// TIA Portal V17 export
// export: Created 2023-02-14T02:49:50.4456623Z, ExportSetting WithDefaults, DisplayName Totally Integrated Automation Portal, DisplayVersion V17, DisplayName TIA Portal Openness, DisplayVersion V17, DisplayName TIA Portal Teamcenter Gateway, DisplayVersion V17, DisplayName TIA Portal Version Control Interface, DisplayVersion V17, DisplayName SINAMICS Startdrive Advanced, DisplayVersion V17, DisplayName SINAMICS Startdrive G130, G150, S120, S150, SINAMICS MV, S210, DisplayVersion V17, DisplayName SINAMICS Startdrive G110M, G120, G120C, G120D, G120P, G115D, DisplayVersion V17, DisplayName STEP 7 Professional, DisplayVersion V17, DisplayName STEP 7 Safety, DisplayVersion V17, DisplayName WinCC Professional, DisplayVersion V17
DATA_BLOCK "T-05.01_DB"   // DB355
VERSION : 0.1
// stored: AutoNumber false, DBAccessibleFromOPCUA true, DBAccessibleFromWebserver true, InstanceOfName BFT_Type2, InstanceOfType FB
"BFT_Type2"
   // VAR_INPUT
   //    "IN_FBAV.01" : Bool;
   //    "IN_FBAV.02" : Bool;
   //    "IN_FBAV.03" : Bool;
   //    "IN_FBAV.04" : Bool;
   //    "IN_FBAV.05" : Bool;
   //    "IN_FBAV.06" : Bool;
   //    "IN_FBAV.07" : Bool;
   //    "IN_FBAV.08" : Bool;
   //    "IN_FBAV.09" : Bool;
   //    "IN_FBAV.10" : Bool;
   //    "IN_FBAV.11" : Bool;
   //    "IN_FBAV.12" : Bool;
   //    IN_LT01 : Real;
   //    "IN_FBP.01" : Bool;
   //    "IN_P.01-Speed" : Real;
   //    "IN_FBP.02" : Bool;
   //    "IN_P.02-Speed" : Real;
   //    "IN_FBP.03" : Bool;
   //    "IN_P.03-Speed" : Real;
   //    IN_FBXA : Bool;
   //    "IN_XA-Speed" : Real;
   //    DosePumpSpeed : Real;
   //    "DoseON-OFF" : Bool;
   //    "DosePumpON-OFF" : Bool;
   //    CIPPulse : Bool;
   //    CIP_Supply_ON : Bool;
   //    CIP_Busy : Bool;
   //    LineTrf_OK : Bool;
   //    LineFlush_OK : Bool;
   //    Loading_Busy : Bool;
   //    LCS_Start : Bool;
   //    LCS_Stop : Bool;
   //    LCS_Dose : Bool;
   //    InloadDose_AV : Bool;
   //    InloadDose_P : Bool;
   //    CountMode : Bool;
   //    FT_Pulse : Bool;
   //    FT_Total : Real;
   //    IN_LDT : Date_And_Time;
   // END_VAR
   // VAR_OUTPUT
   //    "OUT_AV.01" : Bool;
   //    "OUT_AV.02" : Bool;
   //    "OUT_AV.03" : Bool;
   //    "OUT_AV.04" : Bool;
   //    "OUT_AV.05" : Bool;
   //    "OUT_AV.06" : Bool;
   //    "OUT_AV.07" : Bool;
   //    "OUT_AV.08" : Bool;
   //    "OUT_AV.09" : Bool;
   //    "OUT_AV.10" : Bool;
   //    "OUT_AV.11" : Bool;
   //    "OUT_AV.12" : Bool;
   //    "OUT_P.01" : Bool;
   //    "OUT_P.01-Speed" : Real;
   //    "OUT_P.02" : Bool;
   //    "OUT_P.02-Speed" : Real;
   //    "OUT_P.03" : Bool;
   //    "OUT_P.03-Speed" : Real;
   //    OUT_XA : Bool;
   //    "OUT_XA-Speed" : Real;
   //    OUT_InloadDose_Idle : Bool;
   //    OUT_InloadDose_AV : Bool;
   //    OUT_InloadDose_P : Bool;
   //    OUT_InloadDose_P_Speed : Real;
   //    OUT_CIPTank_AVOpen : Bool;
   //    OUT_CIPLine_AVOpen : Bool;
   // END_VAR
   // VAR
   //    Cmd { ExternalAccessible := 'False'; ExternalVisible := 'False'; ExternalWritable := 'False'} : Struct
   //       Inload { ExternalAccessible := 'False'; ExternalVisible := 'False'; ExternalWritable := 'False'} : Bool;
   //       Dose_start { ExternalAccessible := 'False'; ExternalVisible := 'False'; ExternalWritable := 'False'} : Bool;
   //       Dose_pause { ExternalAccessible := 'False'; ExternalVisible := 'False'; ExternalWritable := 'False'} : Bool;
   //       RaadyForMix { ExternalAccessible := 'False'; ExternalVisible := 'False'; ExternalWritable := 'False'} : Bool;
   //       Tank_CIP_Req { ExternalAccessible := 'False'; ExternalVisible := 'False'; ExternalWritable := 'False'} : Bool;
   //       Line_CIP_Req { ExternalAccessible := 'False'; ExternalVisible := 'False'; ExternalWritable := 'False'} : Bool;
   //       Flushing { ExternalAccessible := 'False'; ExternalVisible := 'False'; ExternalWritable := 'False'} : Bool;
   //       Flush_Select { ExternalAccessible := 'False'; ExternalVisible := 'False'; ExternalWritable := 'False'} : Byte;
   //       Agitator_Mode { ExternalAccessible := 'False'; ExternalVisible := 'False'; ExternalWritable := 'False'} : Bool;
   //       Agitator_Man_ONOFF { ExternalAccessible := 'False'; ExternalVisible := 'False'; ExternalWritable := 'False'} : Bool;
   //       Agitator_SpeedMode { ExternalAccessible := 'False'; ExternalVisible := 'False'; ExternalWritable := 'False'} : Bool;
   //    END_STRUCT;
   //    Param { ExternalAccessible := 'False'; ExternalVisible := 'False'; ExternalWritable := 'False'} : Struct
   //       SP_Level_LL { ExternalAccessible := 'False'; ExternalVisible := 'False'; ExternalWritable := 'False'} : Real;
   //       SP_Level_ML { ExternalAccessible := 'False'; ExternalVisible := 'False'; ExternalWritable := 'False'} : Real;
   //       SP_Level_HL { ExternalAccessible := 'False'; ExternalVisible := 'False'; ExternalWritable := 'False'} : Real;
   //       SP_Level_Agi_ON1 { ExternalAccessible := 'False'; ExternalVisible := 'False'; ExternalWritable := 'False'} : Real;
   //       SP_Level_Agi_OFF1 { ExternalAccessible := 'False'; ExternalVisible := 'False'; ExternalWritable := 'False'} : Real;
   //       SP_Level_Agi_ON2 { ExternalAccessible := 'False'; ExternalVisible := 'False'; ExternalWritable := 'False'} : Real;
   //       SP_Level_Agi_OFF2 { ExternalAccessible := 'False'; ExternalVisible := 'False'; ExternalWritable := 'False'} : Real;
   //       SP_Level_Agi_ON3 { ExternalAccessible := 'False'; ExternalVisible := 'False'; ExternalWritable := 'False'} : Real;
   //       SupplyPump_SP_Speed { ExternalAccessible := 'False'; ExternalVisible := 'False'; ExternalWritable := 'False'} : Real;
   //       Agitator_SP_Speed { ExternalAccessible := 'False'; ExternalVisible := 'False'; ExternalWritable := 'False'} : Real;
   //       RawDose_SP_Qty { ExternalAccessible := 'False'; ExternalVisible := 'False'; ExternalWritable := 'False'} : Real;
   //       RawDose_Fine_Qty { ExternalAccessible := 'False'; ExternalVisible := 'False'; ExternalWritable := 'False'} : Real;
   //       RawDose_Stop_Qty { ExternalAccessible := 'False'; ExternalVisible := 'False'; ExternalWritable := 'False'} : Real;
   //       RawDose_SP_Speed { ExternalAccessible := 'False'; ExternalVisible := 'False'; ExternalWritable := 'False'} : Real;
   //       RawDose_Fine_Speed { ExternalAccessible := 'False'; ExternalVisible := 'False'; ExternalWritable := 'False'} : Real;
   //       L_Hi_Lim { ExternalAccessible := 'False'; ExternalVisible := 'False'; ExternalWritable := 'False'} : Real;
   //       L_Lo_Lim { ExternalAccessible := 'False'; ExternalVisible := 'False'; ExternalWritable := 'False'} : Real;
   //       L_Hys { ExternalAccessible := 'False'; ExternalVisible := 'False'; ExternalWritable := 'False'} : Real;
   //       FlushingTime { ExternalAccessible := 'False'; ExternalVisible := 'False'; ExternalWritable := 'False'} : Time;
   //       CIP_Trf_SP_Speed { ExternalAccessible := 'False'; ExternalVisible := 'False'; ExternalWritable := 'False'} : Real;
   //       CIP_Ret_ON_SP { ExternalAccessible := 'False'; ExternalVisible := 'False'; ExternalWritable := 'False'} : Real;
   //       CIP_Ret_OFF_SP { ExternalAccessible := 'False'; ExternalVisible := 'False'; ExternalWritable := 'False'} : Real;
   //    END_STRUCT;
   //    State { ExternalAccessible := 'False'; ExternalVisible := 'False'; ExternalWritable := 'False'} : Struct
   //       Tank_inloading { ExternalAccessible := 'False'; ExternalVisible := 'False'; ExternalWritable := 'False'} : Bool;
   //       Tank_inRawDose { ExternalAccessible := 'False'; ExternalVisible := 'False'; ExternalWritable := 'False'} : Bool;
   //       Tank_inCIP { ExternalAccessible := 'False'; ExternalVisible := 'False'; ExternalWritable := 'False'} : Bool;
   //       Line_inCIP { ExternalAccessible := 'False'; ExternalVisible := 'False'; ExternalWritable := 'False'} : Bool;
   //       Flushing { ExternalAccessible := 'False'; ExternalVisible := 'False'; ExternalWritable := 'False'} : Bool;
   //       Tank_LL { ExternalAccessible := 'False'; ExternalVisible := 'False'; ExternalWritable := 'False'} : Bool;
   //       Tank_ML { ExternalAccessible := 'False'; ExternalVisible := 'False'; ExternalWritable := 'False'} : Bool;
   //       Tank_HL { ExternalAccessible := 'False'; ExternalVisible := 'False'; ExternalWritable := 'False'} : Bool;
   //       L_Agi_ON1 { ExternalAccessible := 'False'; ExternalVisible := 'False'; ExternalWritable := 'False'} : Bool;
   //       L_Agi_ON2 { ExternalAccessible := 'False'; ExternalVisible := 'False'; ExternalWritable := 'False'} : Bool;
   //       L_Agi_ON3 { ExternalAccessible := 'False'; ExternalVisible := 'False'; ExternalWritable := 'False'} : Bool;
   //       Inload_Enable { ExternalAccessible := 'False'; ExternalVisible := 'False'; ExternalWritable := 'False'} : Bool;
   //       Tank_CIP_Enable { ExternalAccessible := 'False'; ExternalVisible := 'False'; ExternalWritable := 'False'} : Bool;
   //       Line_CIP_Enable { ExternalAccessible := 'False'; ExternalVisible := 'False'; ExternalWritable := 'False'} : Bool;
   //       Flushing_Enable { ExternalAccessible := 'False'; ExternalVisible := 'False'; ExternalWritable := 'False'} : Bool;
   //       Flush_selected { ExternalAccessible := 'False'; ExternalVisible := 'False'; ExternalWritable := 'False'} : Byte;
   //       CIP_Request_OK { ExternalAccessible := 'False'; ExternalVisible := 'False'; ExternalWritable := 'False'} : Bool;
   //       CIP_ReturnON { ExternalAccessible := 'False'; ExternalVisible := 'False'; ExternalWritable := 'False'} : Bool;
   //       Ready_For_Transfer_EN { ExternalAccessible := 'False'; ExternalVisible := 'False'; ExternalWritable := 'False'} : Bool;
   //       Ready_For_Transfer { ExternalAccessible := 'False'; ExternalVisible := 'False'; ExternalWritable := 'False'} : Bool;
   //       Transfer_to_Blend { ExternalAccessible := 'False'; ExternalVisible := 'False'; ExternalWritable := 'False'} : Bool;
   //       HWT_Status { ExternalAccessible := 'False'; ExternalVisible := 'False'; ExternalWritable := 'False'} : Int;
   //    END_STRUCT;
   //    alwaysON : Bool;
   //    L_Hys_Abs : Real;
   //    Hys_Level_HL : Real;
   //    Hys_Level_ML : Real;
   //    Hys_Level_LL : Real;
   //    RawDose_Stop_Qty : Real;
   //    "FT Counter" : Real;
   //    "Pulse/Liter" : Real;
   //    AwalTolaizer { S7_SetPoint := 'True'} : Real;
   //    AkhirTolaizer : Real;
   //    TargetTotalizer : Real;
   //    r : Struct
   //       PosE1 : Bool;
   //       PosE2 : Bool;
   //       PosE3 : Bool;
   //       PosE4 : Bool;
   //       PosE5 : Bool;
   //       PosE6 : Bool;
   //       PosE7 : Bool;
   //       PosE8 : Bool;
   //       PosE9 : Bool;
   //       PosE10 : Bool;
   //       PosE11 : Bool;
   //       PosE12 : Bool;
   //       PosE13 : Bool;
   //       PosE14 : Bool;
   //       PosE15 : Bool;
   //       PosE16 : Bool;
   //       PosE17 : Bool;
   //       PosE18 : Bool;
   //       PosE19 : Bool;
   //       PosE20 : Bool;
   //       PosE21 : Bool;
   //       PosE22 : Bool;
   //       PosE23 : Bool;
   //       PosE24 : Bool;
   //       PosE25 : Bool;
   //       PosE26 : Bool;
   //       PosE27 : Bool;
   //       PosE28 : Bool;
   //       PosE29 : Bool;
   //       PosE30 : Bool;
   //       PosE31 : Bool;
   //       PosE32 : Bool;
   //    END_STRUCT;
   //    Actuator : Struct
   //       AV_Outlet : Bool;
   //       TransferPump : Bool;
   //       FlushPump : Bool;
   //       CV_Steam : Bool;
   //       Pump : Bool;
   //       Agitator_level : Bool;
   //       LCS_OnOff : Bool;
   //    END_STRUCT;
   //    FlushingTim : TON_TIME;
   //    SPumpTim { S7_SetPoint := 'True'} : TON_TIME;
   //    AVinloadTim { S7_SetPoint := 'True'} : TON_TIME;
   //    L_AgiTim { S7_SetPoint := 'True'} : TON_TIME;
   //    Dose { S7_SetPoint := 'True'} : "DOSE";
   // END_VAR
BEGIN
END_DATA_BLOCK
